% RSLogix 500 project TEST BB_BAK000.RSS, saved by version 11.00.00.00 %
PROJECT "UNTITLED"    % processor: type code 8 %

PROGRAM FILES
  LAD 2   2 rungs

DATA FILES
  O0 OUTPUT  2 elements
  I1 INPUT  3 elements
  S2 STATUS  16 elements
  B3 BINARY  1 elements
  T4 TIMER  1 elements
  C5 COUNTER  1 elements
  R6 CONTROL  1 elements
  N7 INTEGER  1 elements

LADDER 2
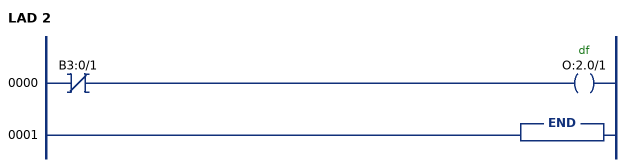
% Rung: 0 %
SOR XIO B3:0/1 OTE O:2.0/1 EOR
%   O:2.0/1  "df" %
% Rung: 1 %
SOR END EOR
